FOR i := 1 TO MAX_TASKS DO
    StatusMessage.Status.Tasks[i].State           := TO_STRING(_Tasks[i].Task.Info.State);
    StatusMessage.Status.Tasks[i].CurrentTaskId   := _Tasks[i].Task.Info.CurrentTaskId;
    StatusMessage.Status.Tasks[i].LineNumber      := _Tasks[i].Task.Info.LineNumber;
    StatusMessage.Status.Tasks[i].StationName     := _Tasks[i].Task.Info.StationName;
    StatusMessage.Status.Tasks[i].SubStation      := _Tasks[i].Task.Info.SubStation;
    StatusMessage.Status.Tasks[i].TotalTaskSteps  := _Tasks[i].Task.Info.TotalTaskSteps;
    StatusMessage.Status.Tasks[i].CurrentTaskStep := _Tasks[i].Task.Info.CurrentTaskStep;
END_FOR;

//Removing for now as SAM doesn't do anything with this information at the moment but has potential in the future
// // Assign values to the Alerts array
// // Alert 1
// i := 1;
// StatusMessage.Status.Alerts[i].Level := 'WARNING';
// StatusMessage.Status.Alerts[i].Message := 'NoPlates';
// 
// // Alert 2
// i := 2;
// StatusMessage.Status.Alerts[i].Level := 'ERROR';
// StatusMessage.Status.Alerts[i].Message := 'Garrick';

// Build the JSON payload
fbJson.ResetDocument();
fbJsonDataType.AddJsonValueFromSymbol(fbJson, 'ST_Messages', SIZEOF(StatusMessage), ADR(StatusMessage));

// Copy the JSON document into sPayload
fbJson.CopyDocument(sPayload, SIZEOF(sPayload));

nPayloadLength    := LEN2(ADR(sPayload));
nLENofPayloadSize := LEN(UDINT_TO_STRING(nPayloadLength));
sLENofPayloadSize := UDINT_TO_STRING(nPayloadLength);

(* Construct the full message with headers and footers using CONCAT2 *)
sRequestMessage := '';
CONCAT2(ADR(sRequestMessage), ADR(MESSAGE_START), ADR(sRequestMessage), SIZEOF(sRequestMessage));
CONCAT2(ADR(sRequestMessage), ADR(PROTOCOL_VERSION), ADR(sRequestMessage), SIZEOF(sRequestMessage));
sTempPayload := 'JSON  ';
CONCAT2(ADR(sRequestMessage), ADR(sTempPayload), ADR(sRequestMessage), SIZEOF(sRequestMessage));
sTempPayload := REPLACE('000000000000', sLENofPayloadSize, nLENofPayloadSize, 13 - nLENofPayloadSize);
CONCAT2(ADR(sRequestMessage), ADR(sTempPayload), ADR(sRequestMessage), SIZEOF(sRequestMessage));
sTempPayload := '  ';
CONCAT2(ADR(sRequestMessage), ADR(sTempPayload), ADR(sRequestMessage), SIZEOF(sRequestMessage));
//Add Payload in
CONCAT2(ADR(sRequestMessage), ADR(sPayload), ADR(sRequestMessage), SIZEOF(sRequestMessage));
sTempPayload := '>>>endOfPacket__';
CONCAT2(ADR(sRequestMessage), ADR(sTempPayload), ADR(sRequestMessage), SIZEOF(sRequestMessage));

ComposeStatus := sRequestMessage;
END_METHOD

METHOD PROTECTED CreateEvents
VAR_INPUT
END_VAR
// Add your event creation here

// Super call to base

SUPER^.CreateEvents();
END_METHOD

METHOD CyclicLogic
VAR_INPUT
END_VAR
IF NOT _InitComplete THEN
    _InitComplete := Initialize();
    RETURN;
END_IF

SUPER^.CyclicLogic();

(* On PLC reset or program download close all old (opened) connections *)

fbCloseAll(sSrvNetID := sSrvNetID, bExecute := _InitComplete);

IF fbCloseAll.bBusy OR fbCloseAll.bError THEN
    RETURN;
END_IF

//fbClient(sSrvNetId := sSrvNetID, bEnable := bEnable, bLog := bLog);

(*-------------------------- Trigger data exchange -----------------------------------------------*)

fbConnection(sSrvNetID   := sSrvNetID,
             fbRx        := fbRx,
             fbTx        := fbTx,
             fbLog       := fbLog,
             bEnable     := bEnable,
             sRemoteHost := SERVER_IP,
             nRemotePort := SERVER_PORT,
             bLog        := bLog,
             sPrefix     := sPrefix,
             eState      => eState);

IF fbConnection.eState = eSOCKET_CONNECTED THEN (* Connection established *)
    Application();
    //fbApplication( fbTx := fbTx, fbRx := fbRx, fbLog := fbLog );
END_IF
END_METHOD

METHOD ExtractMetaData : STRING
VAR_INPUT
    sInputString : STRING; // The string to search within
    sTag         : STRING; // The metadata tag to find
END_VAR

VAR
    iPosTag        : INT;
    iPosValueStart : INT;
    iPosValueEnd   : INT;
    iValueLength   : INT;
    sValue         : STRING[20]; // Adjust size based on expected number length
    c              : BYTE;
    testn          : INT := 1;
END_VAR
// Initialize return value
ExtractMetaData := ''; // Default value if not found or error
c               := sInputString[testn];
// Find the position of the tag in the input string
iPosTag := FIND(sInputString, sTag);

IF iPosTag <> 0 THEN
    // Position where the value starts (immediately after the tag)
    iPosValueStart := iPosTag + LEN(sTag);

    // Initialize iPosValueEnd to the start position
    iPosValueEnd := iPosValueStart;

    // Loop to find the end of the numeric value
    WHILE (iPosValueEnd <= LEN(sInputString)) DO
        c := sInputString[iPosValueEnd];

        IF c <> F_ToASC('$N') THEN
            // It's not EOL, continue
            iPosValueEnd := iPosValueEnd + 1;
        ELSE
            // EOL found
            EXIT;
        END_IF
    END_WHILE

    // Calculate the length of the numeric value
    iValueLength := iPosValueEnd - iPosValueStart + 1;

    IF iValueLength > 0 THEN
        // Extract the numeric value as a string
        sValue := MID(sInputString, iValueLength, iPosValueStart);

        // Convert the string to an integer
        ExtractMetaData := sValue;
    ELSE
        // No numeric value found after the tag
        ExtractMetaData := ''; // Or handle as needed
    END_IF
ELSE
    // Tag not found
    ExtractMetaData := ''; // Or handle as needed
END_IF
END_METHOD

METHOD GenUUID : STRING[32]
VAR_INPUT
END_VAR

VAR
    uuid_str      : STRING[32];
    alpha_numeric : STRING[17] := '0123456789ABCDEF';
    i             : INT;
    Seed          : INT;
    Random        : DRAND;
    rnum          : INT;
END_VAR
(* Generate UUID *)
FOR i := 1 TO 32 DO
    Seed        := TIME_TO_INT(TIME());
    Random.Seed := Seed;
    Random();
    rnum     := LREAL_TO_INT(Random.Num * 16);
    uuid_str := CONCAT(uuid_str, MID(alpha_numeric, 1, rnum));
END_FOR

GenUUID := uuid_str;
END_METHOD

METHOD InfeedLineNumberCheck : INT
VAR_INPUT
    Alternate    : BOOL;
    PreviousLine : INT;
END_VAR

VAR
    jig2Calc : LREAL;
    jig3Calc : LREAL;
END_VAR
IF UseLineOneOnly = FALSE THEN
    jig2Calc := USINT_TO_LREAL(_OutfeedConveyorStatus_Jig2.Occupied) / UDINT_TO_LREAL(_OutfeedConveyorStatus_Jig2.Total);
    jig3Calc := USINT_TO_LREAL(_OutfeedConveyorStatus_Jig3.Occupied) / UDINT_TO_LREAL(_OutfeedConveyorStatus_Jig3.Total);

    IF Alternate = FALSE THEN
        IF jig2Calc = 1 AND jig3Calc = 1 THEN
            InfeedLineNumberCheck := 0;
        ELSIF jig2Calc = 1 THEN
            InfeedLineNumberCheck := 2;
        ELSIF jig3Calc = 1 THEN
            InfeedLineNumberCheck := 1;
        ELSIF jig2Calc <= jig3Calc THEN
            InfeedLineNumberCheck := 1;
        ELSE
            InfeedLineNumberCheck := 2;
        END_IF
    ELSE
        IF jig2Calc = 1 AND jig3Calc = 1 THEN
            InfeedLineNumberCheck := 0;
        ELSIF jig2Calc = 1 THEN
            InfeedLineNumberCheck := 2;
        ELSIF jig3Calc = 1 THEN
            InfeedLineNumberCheck := 1;
        ELSE
            IF PreviousLine = 1 THEN
                InfeedLineNumberCheck := 2;
            ELSE
                InfeedLineNumberCheck := 1;
            END_IF
        END_IF
    END_IF
ELSE
    InfeedLineNumberCheck := 1;
END_IF
END_METHOD

//! @summary Basic module initialization logic
METHOD PROTECTED Initialize : BOOL;
VAR
    i                        : UDINT;
    varInfo                  : __SYSTEM.VAR_INFO;
    AllSubUnitsInitialized   : BOOL := TRUE;
    AllComponentsInitialized : BOOL := TRUE;
END_VAR

//! @description This method is called by <c>CyclicLogic()</c> as required
Initialize := FALSE;

CASE DescendantSequenceState OF
    0:

        _LogModeChanges         := FALSE;
        _LogStateChanges        := FALSE;
        DescendantSequenceState := DescendantSequenceState + 10;

    10:
        //CreateTask('Infeed');

        DescendantSequenceState := DescendantSequenceState + 10;

    20:
        //Copy Mode names

        DescendantSequenceState := DescendantSequenceState + 10;

    30:
        //Call the Super

        IF SUPER^.Initialize() THEN
            DescendantSequenceState := DescendantSequenceState + 10;
        END_IF

    40:
        Initialize := TRUE;
END_CASE
END_METHOD

METHOD IsIdleTask : BOOL
VAR_INPUT
    State : E_TaskState;
END_VAR
IF State = E_TaskState.ACTIVE OR State = E_TaskState.PENDING OR State = E_TaskState.RECOVERY THEN
    IsIdleTask := FALSE;
ELSE
    IsIdleTask := TRUE;
END_IF
END_METHOD

PROPERTY OutfeedConveyorStatus_Jig2 : ST_OutfeedConveyorStatus
SET
_OutfeedConveyorStatus_Jig2 := OutfeedConveyorStatus_Jig2;
END_SET
END_PROPERTY

PROPERTY OutfeedConveyorStatus_Jig3 : ST_OutfeedConveyorStatus
SET
_OutfeedConveyorStatus_Jig3 := OutfeedConveyorStatus_Jig3;
END_SET
END_PROPERTY

METHOD ParseCSVData
VAR_IN_OUT
    Task : ST_Task;
END_VAR

VAR
    CSV           : ST_CSV_Generic;
    FileContent   : STRING[25000];
    Line          : STRING[255];
    FileLine      : STRING[255];
    LineIndex     : INT := 1;
    i             : UDINT;
    commaPos      : UDINT;
    endPos        : UDINT;
    newlinePos    : INT;
    ParsingStep   : UDINT;
    ParsingDetail : UDINT;
END_VAR
// Initialize FileContent with the raw string
FileContent := Task.Data;
MEMSET(ADR(CSV), 0, SIZEOF(CSV));

// Loop until all lines are processed
WHILE (LEN(FileContent) > 0) DO
    // Find the position of '$N' to identify the end of a line
    newlinePos := FIND(FileContent, '$N');

    IF newlinePos > 0 THEN
        // Extract the line including the '$N' marker
        Line := LEFT(FileContent, newlinePos);

        // Remove the processed line from FileContent

        MEMMOVE(ADR(FileContent), ADR(FileContent[newlinePos]), SIZEOF(FileContent)); (* Move/shift remaining bytes in buffer *)

    //FileContent := REPLACE(FileContent, '', 1, newlinePos + LEN('$N'));
    ELSE
        // If no '$N' is found, take the rest as the last line
        Line        := FileContent;
        FileContent := '';
    END_IF

    // Skip empty lines or lines that only contain '$N' or Comment lines (!!)
    IF (LEN(Line) = 0) OR (Line = '$N') OR FIND(Line, '!!') > 0 THEN
        CONTINUE;
    END_IF

    // Prepare to parse the details in the line
    FileLine := Line;

    // Loop to extract up to MAX_DATA_COUNT details separated by commas
    FOR i := 1 TO MAX_DATA_COUNT DO
        commaPos := FIND2(ADR(FileLine), ADR(','));
        endPos   := FIND2(ADR(FileLine), ADR('$N'));

        IF commaPos > 0 THEN
            // Copy the detail up to the comma into your CSV structure
            MEMCPY(ADR(CSV.CSVLines[LineIndex].Fields[i]), ADR(FileLine), commaPos - 1);

            // Remove the extracted detail from FileLine
            MEMMOVE(ADR(FileLine), ADR(FileLine[commaPos]), SIZEOF(FileLine)); (* Move/shift remaining bytes in buffer *)
        ELSIF endPos > 0 THEN
            // Copy the last detail (no more commas found)
            MEMCPY(ADR(CSV.CSVLines[LineIndex].Fields[i]), ADR(FileLine), endPos - 1);
            EXIT; // Exit the loop since there are no more details
        END_IF

    END_FOR

    //Inject into CSV Step Structure
    IF CSV.CSVLines[LineIndex].Fields[1] = 'SeqStart' THEN
        ParsingStep                             := STRING_TO_UDINT(CSV.CSVLines[LineIndex].Fields[3]);
        Task.CSV.Steps[ParsingStep].seqID       := ParsingStep;
        Task.CSV.Steps[ParsingStep].seqName     := STRING_TO_E_CommandName(CSV.CSVLines[LineIndex].Fields[2]);
        Task.CSV.Steps[ParsingStep].DetailCount := STRING_TO_UDINT(CSV.CSVLines[LineIndex].Fields[4]);
    ELSIF CSV.CSVLines[LineIndex].Fields[1] = 'SeqDetail' THEN
        ParsingDetail                                                := STRING_TO_UDINT(CSV.CSVLines[LineIndex].Fields[2]);
        Task.CSV.Steps[ParsingStep].Details[ParsingDetail].DetailID  := ParsingDetail;
        Task.CSV.Steps[ParsingStep].Details[ParsingDetail].DataCount := STRING_TO_UDINT(CSV.CSVLines[LineIndex].Fields[3]);

        FOR j := 1 TO Task.CSV.Steps[ParsingStep].Details[ParsingDetail].DataCount DO
            Task.CSV.Steps[ParsingStep].Details[ParsingDetail].Datas[j] := CSV.CSVLines[LineIndex].Fields[j + 3];
        END_FOR
    ELSIF CSV.CSVLines[LineIndex].Fields[1] = 'SeqEnd' THEN
        Task.Info.TotalTaskSteps := STRING_TO_DINT(CSV.CSVLines[LineIndex].Fields[3]);
    END_IF

    // Move to the next line index
    LineIndex := LineIndex + 1;
END_WHILE
END_METHOD

METHOD ProcessReceivedMessage : BOOL
VAR_INPUT
    sReceiveData : STRING[25000];
END_VAR

VAR
    nPayloadLength    : INT;
    nLENofPayloadSize : INT;
    sPayloadSize      : STRING(36);
    sMessageBody      : STRING[25000];
    uuid_str          : STRING(36);
    fbTime            : FB_LocalSystemTime := (bEnable := TRUE);
    currentDateTime   : DATE_AND_TIME;
    eContentType      : E_ContentType; (* Enum for message content type *)
    sMessageCategory  : STRING(20); (* JSON Message Category *)
    eMessageCategory  : E_MessageCategory; (* Enum for message category *)
    sInResponseToUuid : STRING(36); (* JSON InResponseToUuid *)

    fbJson   : FB_JsonDomParser;
    jsonRoot : SJsonValue;
    jsonProp : SJsonValue;

    jig2Calc : LREAL;
    jig3Calc : LREAL;

END_VAR
(* Determine message type and set enum value *)

MEMSET(ADR(sMessageBody), 0, SIZEOF(sMessageBody));

IF FIND2(ADR(sReceiveData), ADR('JSON'),) > 0 THEN
    eContentType := E_ContentType.CT_JSON;
    MEMCPY(ADR(sPayloadSize), ADR(sReceiveData[34]), 12);
    MEMCPY(ADR(sMessageBody), ADR(sReceiveData[48]), STRING_TO_UDINT(sPayloadSize));
ELSIF FIND2(ADR(sReceiveData), ADR('ACK'),) > 0 THEN
    eContentType := E_ContentType.CT_JSON;
    MEMCPY(ADR(sPayloadSize), ADR(sReceiveData[34]), 12);
    MEMCPY(ADR(sMessageBody), ADR(sReceiveData[48]), STRING_TO_UDINT(sPayloadSize));
ELSIF FIND2(ADR(sReceiveData), ADR('NOTASK'),) > 0 THEN
    eContentType := E_ContentType.CT_JSON;
    MEMCPY(ADR(sPayloadSize), ADR(sReceiveData[34]), 12);
    MEMCPY(ADR(sMessageBody), ADR(sReceiveData[48]), STRING_TO_UDINT(sPayloadSize));
ELSIF FIND2(ADR(sReceiveData), ADR('CSV')) > 0 THEN
    eContentType := E_ContentType.CT_CSV;
    MEMCPY(ADR(sPayloadSize), ADR(sReceiveData[34]), 12);
    MEMCPY(ADR(sMessageBody), ADR(sReceiveData[48]), STRING_TO_UDINT(sPayloadSize));
ELSE
    eContentType           := E_ContentType.CT_NONE;
    ProcessReceivedMessage := FALSE;
    fbLog.Message(sMessage := 'Failed to read Content type of Message from SAM');
    RETURN;
END_IF

(* Process JSON message *)
IF eContentType = E_ContentType.CT_JSON THEN
    fbJson.ParseDocument(sMessageBody);
    jsonRoot := fbJson.GetDocumentRoot();

    (* Extract Message Category and UUID *)
    jsonProp := fbJson.FindMember(jsonRoot, 'MessageCategory');

    IF (jsonProp <> 0) THEN
        sMessageCategory := fbJson.GetString(jsonProp);
    END_IF

    jsonProp := fbJson.FindMember(jsonRoot, 'InResponseToUuid');

    IF (jsonProp <> 0) THEN
        sInResponseToUuid := fbJson.GetString(jsonProp);
    END_IF

    (* Set the message category enum based on extracted value using FIND *)
    IF sMessageCategory = 'RequestForInfo' THEN
        eMessageCategory       := E_MessageCategory.MC_RFI;
        ProcessReceivedMessage := TRUE;
    ELSIF sMessageCategory = 'Info' THEN
        eMessageCategory := E_MessageCategory.MC_INFO;
        fbLog.Message(sMessage := 'RFI message response received.');
        Trace(CONCAT('RFI message response received: Task # -> ', INT_TO_STRING(RFT_Index)));
        ProcessReceivedMessage := TRUE;
    ELSIF sMessageCategory = 'Task' THEN
        eMessageCategory := E_MessageCategory.MC_TASK;
        fbLog.Message(sMessage := 'TASK message response received.');
        Trace(CONCAT('TASK message response received: Task # -> ', INT_TO_STRING(RFT_Index)));
        ProcessReceivedMessage := TRUE;
    ELSIF sMessageCategory = 'NoTask' = 1 THEN
        eMessageCategory                     := E_MessageCategory.MC_NOTASK;
        _Tasks[RFT_Index].Task.RFT_Requested := FALSE;
        //indexing to next task due to no task being received for current
        IF RFT_Index = 1 THEN
            _Tasks[RFT_Index].Task.Info.State := E_TaskState.IDLE;
            InfeedPreviousLineRequest         := _Tasks[RFT_Index].Task.Info.LineNumber;
            InfeedAlternateLine               := TRUE;
        END_IF

        ProcessReceivedMessage := TRUE;

        fbLog.Message(sMessage := 'NOTASK message response received.');
        Trace(CONCAT('NOTASK message response received: Task # -> ', INT_TO_STRING(RFT_Index)));
        Trace(CONCAT('NOTASK message response for Line number -> ', INT_TO_STRING(_Tasks[RFT_Index].Task.Info.LineNumber)));
    ELSIF sMessageCategory = 'Status' THEN
        eMessageCategory       := E_MessageCategory.MC_STATUS;
        ProcessReceivedMessage := TRUE;
    ELSIF sMessageCategory = 'StatusAck' THEN
        eMessageCategory := E_MessageCategory.MC_STATUS_ACK;
        fbLog.Message(sMessage := 'STATUS ACK message response received.');
        Trace(CONCAT('STATUS ACK message response received: Task # -> ', INT_TO_STRING(RFT_Index)));
        // 
        //         IF CurrentMessageUID = sInResponseToUuid THEN
        //             //Success!
        //             ProcessReceivedMessage := TRUE;
        //         ELSE
        //             //No Success!
        //             ProcessReceivedMessage := FALSE;
        //         END_IF
        ProcessReceivedMessage := TRUE;
    ELSIF sMessageCategory = 'NAK' THEN
        eMessageCategory := E_MessageCategory.MC_NAK;
        fbLog.Message(sMessage := 'STATUS NOT ACK message response received.');
        Trace(CONCAT('STATUS NOT ACK message response received: Task # -> ', INT_TO_STRING(RFT_Index)));
        ProcessReceivedMessage := TRUE;
    ELSE
        eMessageCategory       := E_MessageCategory.MC_NONE;
        ProcessReceivedMessage := TRUE;
    END_IF
ELSIF eContentType = E_ContentType.CT_CSV THEN
    //ParseCSV Here

    IF NOT IsIdleTask(_Tasks[RFT_Index].Task.Info.State) THEN
        //if duplicate CSV is recieved when the task is running, ignore new task and keep running old one.
        Trace(CONCAT('Data Parsed for ActiveTask: Task # -> ', INT_TO_STRING(RFT_Index)));
        ProcessReceivedMessage := TRUE;
    ELSE
        _Tasks[RFT_Index].Task.Data               := sMessageBody;
        _Tasks[RFT_Index].Task.Info.CurrentTaskId := STRING_TO_UDINT(ExtractMetaData(sInputString := sMessageBody, sTag := 'SAM Task Id:'));
        ParseCSVData(Task := _Tasks[RFT_Index].Task);

        ProcessReceivedMessage            := TRUE;
        _Tasks[RFT_Index].Task.Info.State := E_TaskState.PENDING;
        Trace(CONCAT('CSV parsed from ProcessReceivedMessage: Task # -> ', INT_TO_STRING(RFT_Index)));
        Trace(CONCAT('CSV parsed for Line number -> ', INT_TO_STRING(_Tasks[RFT_Index].Task.Info.LineNumber)));
    END_IF

    _Tasks[RFT_Index].Task.RFT_Requested := FALSE;

    //     IF CurrentMessageUID = sInResponseToUuid THEN
    //         //Success!
    //         ProcessReceivedMessage            := TRUE;
    //         _Tasks[RFT_Index].Task.Info.State := E_TaskState.PENDING;
    //         fbLog.Error(sMessage := 'CSV parsed from ProcessReceivedMessage');
    //     ELSE
    //         //No Success!
    //         ProcessReceivedMessage := FALSE;
//     END_IF
END_IF
END_METHOD

METHOD RaiseAlarm2Args
VAR_IN_OUT
    fbAlarm : FB_TcAlarm; //Alarm to be raised
END_VAR

VAR_INPUT
    String_1 : STRING; //First String Parameter (The Name of this component will be applied first automatically)
    String_2 : STRING; //Second String Parameter
END_VAR
F_RaiseAlarmWithStringParameters(Alarm := fbAlarm, String_1 := Name, String_2 := String_1, String_3 := String_2);
END_METHOD

METHOD STRING_TO_E_CommandName : E_CommandName
VAR_INPUT
    Name : STRING;
END_VAR
IF Name = 'AssemblyStart' THEN
    STRING_TO_E_CommandName := E_CommandName.AssemblyStart;
ELSIF Name = 'TrussInfo' THEN
    STRING_TO_E_CommandName := E_CommandName.TrussInfo;
ELSIF Name = 'PuckMove' THEN
    STRING_TO_E_CommandName := E_CommandName.PuckMove;
ELSIF Name = 'PickPlace' THEN
    STRING_TO_E_CommandName := E_CommandName.PickPlace;
ELSIF Name = 'ManualBoard' THEN
    STRING_TO_E_CommandName := E_CommandName.ManualBoard;
ELSIF Name = 'BoardInfo' THEN
    STRING_TO_E_CommandName := E_CommandName.BoardInfo;
ELSIF Name = 'Board' THEN
    STRING_TO_E_CommandName := E_CommandName.Board;
ELSIF Name = 'NailPlate' THEN
    STRING_TO_E_CommandName := E_CommandName.NailPlate;
ELSIF Name = 'IndexConveyor' THEN
    STRING_TO_E_CommandName := E_CommandName.IndexConveyor;
ELSIF Name = 'ManualPlate' THEN
    STRING_TO_E_CommandName := E_CommandName.ManualPlate;
ELSIF Name = 'AssemblyEnd' THEN
    STRING_TO_E_CommandName := E_CommandName.AssemblyEnd;
ELSE
    // Handle unknown command name

    STRING_TO_E_CommandName := E_CommandName.Unknown;
END_IF
END_METHOD

PROPERTY Tasks : ARRAY[1..MAX_TASKS] OF ST_TaskREF;
SET
_Tasks := Tasks;
END_SET
END_PROPERTY

END_FUNCTION_BLOCK

// ---- Machine/HMI Connections/FB_ControlSource_MBI.TcPOU
FUNCTION_BLOCK FB_ControlSource_MBI EXTENDS FB_CyclicFB IMPLEMENTS I_PackML_ExternalController
VAR_INPUT
END_VAR

VAR_OUTPUT
END_VAR

VAR
    ipModule                  : I_PackML_Control;
    MainPMLControl_Simplified : ST_PackML_Control_Simplified;
    MainPMLControl_Standard   : ST_PackML_Control;
    R_HMICommand              : R_TRIG;

    MBI_IdleMode        : BOOL;
    MBI_AutoMode AT %I* : BOOL;
    MBI_Manual1  AT %I* : BOOL;
    MBI_Manual2  AT %I* : BOOL;
END_VAR

PROPERTY Control : SPT_BaseTypes.I_PackML_Control
SET
ipModule := Control;
END_SET
END_PROPERTY

METHOD CyclicLogic
VAR
    i : UDINT;
END_VAR
IF NOT _InitComplete THEN
    _InitComplete := Initialize();
    RETURN;
END_IF

MainPMLControl_Standard.CurrentMode  := ipModule.CurrentMode;
MainPMLControl_Standard.CurrentState := ipModule.CurrentState;

FOR i := 1 TO 5 DO
    MainPMLControl_Standard.ModeNames[i] := F_UnitModeToString(UDINT_TO_DINT(i));
END_FOR

MBI_IdleMode := (NOT MBI_AutoMode) AND (NOT MBI_Manual1) AND (NOT MBI_Manual2);

IF MBI_IdleMode THEN
    //Process HMI requests
    R_HMICommand(CLK := (MainPMLControl_Simplified.ResetPressed XOR MainPMLControl_Simplified.StartPressed XOR MainPMLControl_Simplified.StopPressed
                            ) XOR
                        (MainPMLControl_Standard.StateCommand <> E_PMLCommand.ePMLCommand_Undefined AND
                        ipModule.StateCommand <> MainPMLControl_Standard.StateCommand) XOR
                        (ipModule.ModeCommand <> MainPMLControl_Standard.ModeCommand));

END_IF

IF R_HMICommand.Q THEN
    IF MainPMLControl_Simplified.ResetPressed AND
       MainPMLControl_Simplified.ResetPermissive AND
       MainPMLControl_Standard.CurrentState = E_PMLState.ePMLState_Aborted THEN
        ipModule.ChangeState(Tc3_PackML_V2.E_PMLCommand.ePMLCommand_Clear);
    ELSIF MainPMLControl_Simplified.ResetPressed AND MainPMLControl_Simplified.ResetPermissive THEN
        ipModule.ChangeState(Tc3_PackML_V2.E_PMLCommand.ePMLCommand_Reset);
    ELSIF MainPMLControl_Simplified.StartPressed AND MainPMLControl_Simplified.StartPermissive THEN
        IF MainPMLControl_Standard.CurrentState = Tc3_PackML_V2.E_PMLState.ePMLState_Idle THEN
            ipModule.ChangeState(Tc3_PackML_V2.E_PMLCommand.ePMLCommand_Start);
        ELSIF MainPMLControl_Standard.CurrentState = Tc3_PackML_V2.E_PMLState.ePMLState_Held THEN
            ipModule.ChangeState(Tc3_PackML_V2.E_PMLCommand.ePMLCommand_Unhold);
        ELSIF MainPMLControl_Standard.CurrentState = Tc3_PackML_V2.E_PMLState.ePMLState_Suspended THEN
            ipModule.ChangeState(Tc3_PackML_V2.E_PMLCommand.ePMLCommand_Unsuspend);
        END_IF
    ELSIF MainPMLControl_Simplified.StopPressed AND MainPMLControl_Simplified.StopPermissive THEN
        ipModule.ChangeState(Tc3_PackML_V2.E_PMLCommand.ePMLCommand_Hold);
    ELSIF ipModule.StateCommand <> MainPMLControl_Standard.StateCommand THEN
        ipModule.StateCommand := MainPMLControl_Standard.StateCommand;
    ELSIF ipModule.ModeCommand <> MainPMLControl_Standard.ModeCommand THEN
        ipModule.ModeCommand := MainPMLControl_Standard.ModeCommand;
    END_IF
END_IF

MainPMLControl_Simplified.StartPermissive := MainPMLControl_Standard.CurrentState = Tc3_PackML_V2.E_PMLState.ePMLState_Idle OR
                                             MainPMLControl_Standard.CurrentState = Tc3_PackML_V2.E_PMLState.ePMLState_Held OR
                                             MainPMLControl_Standard.CurrentState = Tc3_PackML_V2.E_PMLState.ePMLState_Suspended;

MainPMLControl_Simplified.StopPermissive := MainPMLControl_Standard.CurrentState = Tc3_PackML_V2.E_PMLState.ePMLState_Execute;

MainPMLControl_Simplified.ResetPermissive := MainPMLControl_Standard.CurrentState = Tc3_PackML_V2.E_PMLState.ePMLState_Complete OR
                                             MainPMLControl_Standard.CurrentState = Tc3_PackML_V2.E_PMLState.ePMLState_Stopped OR
                                             MainPMLControl_Standard.CurrentState = Tc3_PackML_V2.E_PMLState.ePMLState_Aborted;
END_METHOD

METHOD FINAL Initialize : BOOL
IF Registered THEN
    Initialize := TRUE;
END_IF
END_METHOD

METHOD FINAL ModeChanged
VAR_INPUT
    NewMode : SPT_BaseTypes.E_PMLUnitMode;
END_VAR
MainPMLControl_Standard.ModeCommand := NewMode;
END_METHOD

PROPERTY Registered : BOOL
GET
Registered := ipModule <> 0;
END_GET
END_PROPERTY

METHOD FINAL StateChanged
VAR_INPUT
    NewState : SPT_BaseTypes.E_PMLCommand;
END_VAR
MainPMLControl_Standard.StateCommand := NewState;
END_METHOD

END_FUNCTION_BLOCK

// ---- Machine/HMI Connections/FB_ControlSource_HMI_Machine.TcPOU
FUNCTION_BLOCK FB_ControlSource_HMI_Machine EXTENDS FB_ControlSource_HMI
VAR_INPUT
END_VAR

VAR_OUTPUT
END_VAR

VAR
END_VAR

METHOD CyclicLogic
VAR_INPUT
END_VAR
SUPER^.CyclicLogic();

//Change the start permissive for the Machine 
MainPMLControl_Simplified.StartPermissive := MainPMLControl_Standard.CurrentState = Tc3_PackML_V2.E_PMLState.ePMLState_Idle OR
                                             (MainPMLControl_Standard.CurrentState = Tc3_PackML_V2.E_PMLState.ePMLState_Held);
END_METHOD

END_FUNCTION_BLOCK

// ---- Project Information/F_GetCompany.TcPOU
// This function has been automatically generated from the project information.
{attribute 'signature_flag' := '1073741824'}
{attribute 'TcGenerated'}
{attribute 'no-analysis'}
FUNCTION F_GetCompany : WSTRING
VAR_INPUT
	
END_VAR

F_GetCompany := "Sawtooth Robotics";

END_FUNCTION

// ---- Project Information/F_GetTitle.TcPOU
// This function has been automatically generated from the project information.
{attribute 'signature_flag' := '1073741824'}
{attribute 'TcGenerated'}
{attribute 'no-analysis'}
FUNCTION F_GetTitle : WSTRING
VAR_INPUT
	
END_VAR

F_GetTitle := "RoofTrussLibrary";

END_FUNCTION

// ---- Project Information/F_GetVersion.TcPOU
// This function has been automatically generated from the project information.
{attribute 'signature_flag' := '1073741824'}
{attribute 'TcGenerated'}
{attribute 'no-analysis'}
FUNCTION F_GetVersion : ST_LibVersion
VAR_INPUT
	
END_VAR

F_GetVersion.iMajor := 0;
F_GetVersion.iMinor := 1;
F_GetVersion.iBuild := 0;
F_GetVersion.iRevision := 0;
F_GetVersion.sVersion := '0.1.0.0';
F_GetVersion.nFlags := 0;

END_FUNCTION

// ---- GlobalTextList.TcGTLO
TEXTLIST GlobalTextList
  733 = '%0.1f °'
  244 = '%i'
  685 = '%s'
  680 = 'Abort'
  842 = 'Async Submodules'
  942 = 'Auto Mode'
  666 = 'AxisInfo'
  452 = 'Clear'
  809 = 'Clear Unwind'
  110 = 'Enabled: %i'
  424 = 'EStop'
  362 = 'File ready for Parse'
  581 = 'Geared: %i'
  744 = 'Hold'
  127 = 'Info Layers'
  625 = 'Load Block Infeed'
  989 = 'Load Board Infeed'
  517 = 'Low Air'
  347 = 'MACHINE'
  46 = 'Maintenance'
  904 = 'Manual'
  312 = 'Pos: %i'
  929 = 'Production'
  181 = 'Reset'
  538 = 'Reset Unwind'
  354 = 'Safety Reset'
  810 = 'Skip Robot Handshakes'
  997 = 'StackLight'
  77 = 'Start'
  804 = 'Start Unwind'
  516 = 'State: %s'
  503 = 'StateComplete'
  289 = 'Step Number'
  828 = 'Stop'
  806 = 'Suspend'
  652 = 'Sync Submodules'
  995 = 'Temp Setpoint'
  197 = 'Unhold'
  832 = 'Unsuspend'
  498 = 'Vel: %i'
END_TEXTLIST
